DATA_BLOCK "GlueningRotaryTable"
{InstructionName := 'BasicPosControl';
 LibVersion := '2.1';
 S7_Optimized_Access := 'TRUE' }
AUTHOR : DRVDPS7
FAMILY : DRIVES
NAME : SINA_POS
VERSION : 5.2
NON_RETAIN
BasicPosControl

BEGIN
   HWIDSTW := 451;
   HWIDZSW := 451;
   srNIST_BFactor := 0.000100582838058472;

END_DATA_BLOCK

